FUNCTION Convert_USINT_TO_ULINT : BOOL
VAR_INPUT
	in : USINT;
	out : REFERENCE TO ULINT;
END_VAR
VAR
	converted : ULINT;
END_VAR

converted := USINT_TO_ULINT(in);

IF (ULINT_TO_USINT(converted) <> in) THEN
	RETURN;
END_IF

out := converted;
Convert_USINT_TO_ULINT := TRUE;

END_FUNCTION

(* stored: Version 1.1.0.1, ProductVersion 3.1.4024.12
   POU Convert_USINT_TO_ULINT: Id {0eb44273-7613-4bda-9b5f-0111de00edeb}, SpecialFunc None *)
